Staubli VAL3: RobotCommandMsg.pjx

--- RobotCommandMsg.pjx ---
Parameters version=s7.7.2 stackSize=5000 millimeterUnit=true
Program file=start.pgx
Program file=stop.pgx
Data file=RobotCommandMsg.dtx
Type name=MessageHeader path=Disk://ros2_server/Types/MessageHeader/MessageHeader.pjx
Type name=RobotCommand path=Disk://ros2_server/Types/RobotCommand/RobotCommand.pjx

--- RobotCommandMsg.dtx ---
public bool bIsInitialized = true
public MessageHeader header
public RobotCommand robotCommand
public num nSerializedData
